(* PLC project Generated.project, CODESYS CODESYS V3.5 SP19 Patch 1 *)
(* stored: creationDateTime 2026-11-18T15:31:54.338901, modificationDateTime 2026-11-18T15:31:54.338901 *)

(* ═══════════════════════════════════════════════════════════════ 🎮 ST_TranslationCmd — Commandes IHM pour la Translation M3 ─────────────────────────────────────────────────────────────── 🎨 Destiné au pilotage de la translation M3 depuis l'IHM. 📄 : Initialized protège SetFreq_Hz (seul réglage à survivre au reboot), sans pont générique pour ne jamais persister BtnTremie/BtnMaintenance. ═══════════════════════════════════════════════════════════════ *)
TYPE ST_TranslationCmd : STRUCT
  SelPositioning : BOOL;  (* 🎯 TRUE = positionneur sur SelTarget ; FALSE = jog libre *)
  SelTarget : INT;  (* 🔢 Numéro de la cible de position sélectionnée *)
  BtnTremie : BOOL;  (* ↔️ Requête marche vers Trémie (ex-BtnFwd), pilotage IHM exclusif *)
  BtnMaintenance : BOOL;  (* ↔️ Requête marche vers Maintenance (ex-BtnRev), pilotage IHM exclusif *)
  SetFreq_Hz : REAL;  (* 🎯 Consigne fréquence manuelle [Hz], limitée par PRG_06_Outputs *)
  InvertDirection : BOOL;  (* 🔀 Switch machine unique : GVL_IHM.Modes.Cmd.TglJoystickMaster (ST_ModesCmd), applicable à M1/M2 ET M3. 🔄 TRUE = inverse Fwd→Maintenance / Rev→Trémie (mise en service) *)
  TglMaintenanceZoneAccess : BOOL;  (* : autorisation CONSCIENTE zone Maintenance, EN PLUS de MAINT_N2 (Auth.MaintenanceM3TargetEnable) *)
  TglAllowWinchMoveAtTremie : BOOL;  (* T249 : autorisation CONSCIENTE montee/descente treuil couple (WinchSel=0) a la Tremie, EN PLUS de la garde WinchSel=2 forcee (FB_Modes) *)
  Initialized : BOOL := FALSE;  (* 🚦 TRUE = SetFreq_Hz restauré depuis GVL_PERSISTENT ce boot *)
  BtnSetAtP1 : BOOL;  (* 🎯 Forcage position P1 depuis IHM en MAINT_N2 (mise en service) *)
END_STRUCT;
END_TYPE
